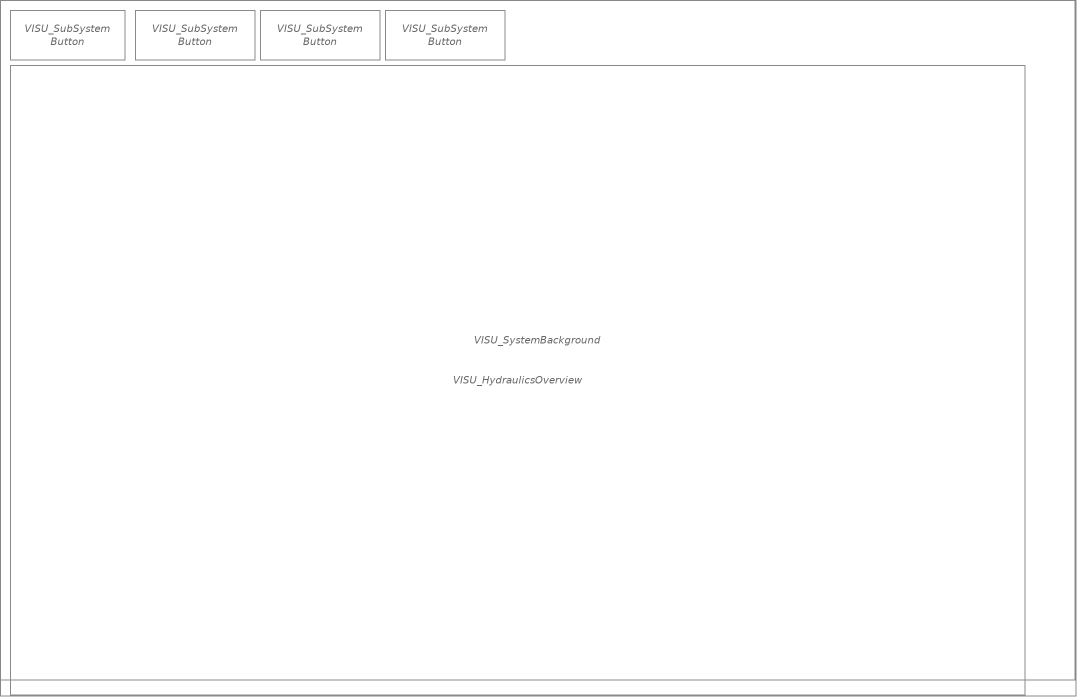
VISUALIZATION VISU_Hydraulics  // 1077x697
VAR_IN_OUT
	ref : Hydraulics;
    widget : HydraulicsWidget;
	ref_safetyHydraulics : SafetyHydraulics;
	ref_safetyIO : SafetyIO;
END_VAR
    Frame (0,0 1075x680)
        shows VISU_SystemBackground(color := widget.actualStatus.color)
    Frame (10,65 1015x630)
        shows VISU_HydraulicsOverview(ref := ref, widget := widget, ref_safety := ref_safetyHydraulics)
        shows VISU_HydraulicsTechnical(ref := ref, widget := widget, ref_safety := ref_safetyHydraulics)
        shows VISU_HydraulicsIO(ref := ref.parts.io, ref_safetyIO := ref_safetyIO, widget := widget.io)
        shows VISU_HydraulicsConfig(editable := ref.editableConfig, active := ref.config, mgr := ref.parts.configManager, mgrWidget := widget.configManager, widget := widget)
        shows VISU_SafetyIO(ref := ref.parts.io, widget := widget.io)
        shows VISU_SafetyConfig(editable := ref.editableConfig, active := ref.config, mgr := ref.parts.configManager, mgrWidget := widget.configManager, widget := widget)
        p701045219: ref.editableConfig
        p2690442461: ref.config
    Frame (10,10 115x50)
        shows VISU_SubSystemButton(widget := widget.button_overview)
        OnMouseClick: FrameSelectionChange Selection=SelectedFrame=b1e9e4b0-bf3d-440f-90c5-cb513105ccf1, GlobSel=AssignType=Directly, SelType=Locally
        OnMouseClick: execute { widget.activeTab := HydraulicsTabs.OVERVIEW; }
    Frame (260,10 120x50)
        shows VISU_SubSystemButton(widget := widget.button_io)
        OnMouseClick: FrameSelectionChange Selection=SelectedFrame=b1e9e4b0-bf3d-440f-90c5-cb513105ccf1, Selection=2, GlobSel=AssignType=Directly, SelType=Locally
        OnMouseClick: execute { widget.activeTab := HydraulicsTabs.IO; }
    Frame (385,10 120x50)
        shows VISU_SubSystemButton(widget := widget.button_config)
        OnMouseClick: FrameSelectionChange Selection=SelectedFrame=b1e9e4b0-bf3d-440f-90c5-cb513105ccf1, Selection=3, GlobSel=AssignType=Directly, SelType=Locally
        OnMouseClick: execute { widget.activeTab := HydraulicsTabs.CONFIG; }
    Frame (135,10 120x50)
        shows VISU_SubSystemButton(widget := widget.button_technical)
        OnMouseClick: FrameSelectionChange Selection=SelectedFrame=b1e9e4b0-bf3d-440f-90c5-cb513105ccf1, Selection=1, GlobSel=AssignType=Directly, SelType=Locally
        OnMouseClick: execute { widget.activeTab := HydraulicsTabs.TECHNICAL; }
END_VISUALIZATION

(* stored: Version 1.1.0.1, ProductVersion 3.1.4019.2
   Visu VISU_Hydraulics: Id {e612f2f3-4460-4b84-aa55-312a8dd3fc38} *)
